FUNCTION_BLOCK PUBLIC FB_ALARM_HANDLER EXTENDS FBA_ALARM_HANDLER
VAR_IN_OUT
	Repository : FBA_ALARM_HANDLER;
END_VAR
VAR_INPUT
	Prefix : STRING;
END_VAR
VAR_OUTPUT
END_VAR
VAR
END_VAR

METHOD RegisterAlarm : REFERENCE TO FBA_ALARM_HANDLER
VAR_INPUT
	Alarm	: REFERENCE TO FB_ALARM;
	Prefix	: STRING := '';
	Update : BOOL := TRUE;
END_VAR
VAR
	TempString : STRING := '';
END_VAR
{warning disable C0371}

// Checking the VAR_IN_OUT reference, leave the current method in case of invalid reference
IF NOT __ISVALIDREF(THIS^.Repository) THEN
     RETURN;
END_IF


IF THIS^.Prefix <> '' THEN
	TempString := CONCAT(THIS^.Prefix, '*');
END_IF;

TempString := CONCAT(TempString, Prefix);
THIS^.Repository.RegisterAlarm(Alarm := Alarm, Prefix := TempString, Update := TRUE);

RegisterAlarm REF= THIS^;
END_METHOD

END_FUNCTION_BLOCK

(* stored: Version 1.1.0.1, ProductVersion 3.1.4024.12
   POU FB_ALARM_HANDLER: Id {6e6866db-2555-4b14-ad23-9aafadc1eed0}, SpecialFunc None
   Method RegisterAlarm: Id {c5b1e60a-b768-4a6b-805f-27263b19fdc9} *)
